RoboDK station: Machine-Tending-Machining-and-Material-Handling-with-Omron-TM12X.rdk

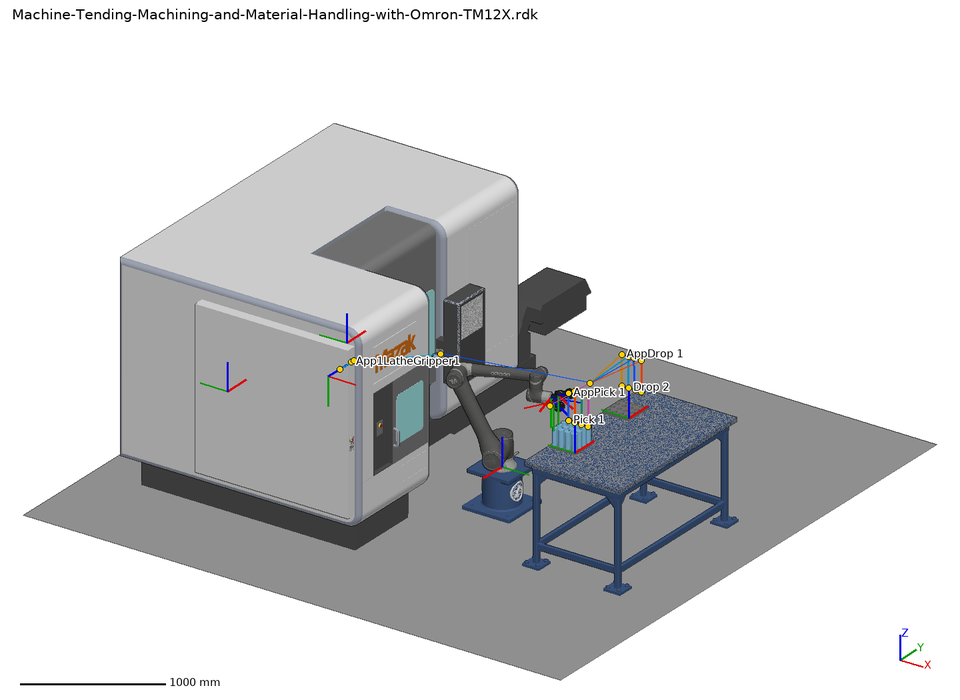
[picture v0: the station drawn from its stored meshes, robots at their saved joint values, targets as dots, program paths as lines]
Station Machine Tending, Machining and Material Handling with Omron TM12X (saved by RoboDK 5.4.3). Poses are relative to the parent item; angles as X-Y-Z fixed-axis rotations.
Station parameters (name, value as stored): TAGS, ['Machine Tending', 'CNC']
  - frame Omron TM12X Base at (300, 0, 70) mm, rotated rx 0 ry 0 rz -90 deg
    - robot Omron TM12X: 6 axes, payload 12 kg, reach 1300 mm, repeatability 0.1 mm, weight 33.3 kg
        modified DH rows (alpha deg, a mm, theta deg, d mm): 0, 0, 0, 165.2; 90, 0, 90, 0; 0, 636.1, 0, 0; 0, 557.9, -90, 156.3; -90, 0, 0, 106; 90, 0, 180, 113.15
        joint limits [-360, -360, -163, -360, -360, -360] to [360, 360, 163, 360, 360, 360]; home [0, 0, 90, -90, 90, 0]; saved at [109.92, -25.7, 113.76, -268.05, -85.72, 0]
      - frame RobotiQ HandE Dual Gripper at (0, 0, -5) mm
        - frame RobotiQ HandE Gripper Base 1 at (50, 0, 40) mm, rotated rx 0 ry 45 rz 0 deg
          - robot RobotiQ HandE Gripper 1: 1 axes
              joint limits [0] to [50]; home [0]; saved at [50]
        - frame RobotiQ HandE Gripper Base 2 at (-50, 0, 40) mm, rotated rx 0 ry -45 rz 0 deg
          - robot RobotiQ HandE Gripper 2: 1 axes
              joint limits [0] to [50]; home [0]; saved at [50]
        - object Hand-E RobotiQ Dual Mounting at (0, 0, 0) mm, size 158.7 x 86.1 x 105 mm, geometry from Hand-E RobotiQ Dual Mounting.step
      - tool Gripper1, TCP at (145, 0, 130) mm, rotated rx 45 ry 0 rz 90 deg
      - tool Gripper2, TCP at (-145, 0, 130) mm, rotated rx -45 ry 0 rz 90 deg
    - object Pedestal H12in (Type 1) at (0, 0, -300) mm, size 400 x 400 x 304.8 mm, geometry from Pedestal-H12in-Type-1.sld
  - frame Mazak Lathe Base at (-1000, 0, 650) mm, rotated rx 0 ry 0 rz 90 deg
    - robot Mazak Lathe: 1 axes
        modified DH rows (alpha deg, a mm, theta deg, d mm): 0, 0, 0, 0 linear
        base shift (0, 0, 0) mm, rotated rx 0 ry 90 rz 0 deg
        joint limits [0] to [700]; home [0]; saved at [0]
    - frame Lathe at (-368.68, -104.77, -79.13) mm, rotated rx -90 ry 0 rz -90 deg
      - target App1LatheGripper1 (Cartesian target) at (-0.18, 0.1, 274.88) mm, rotated rx 0 ry 90 rz 165 deg; joints [287.606, 19.83, 87.712, -318.746, -74.815, 80.984] of Omron TM12X
      - target LatheGripper1 (Cartesian target) at (-0.18, 0.1, 134.88) mm, rotated rx 0 ry 90 rz 165 deg; joints [296.712, 22.07, 84.693, -319.639, -67.09, 75.877] of Omron TM12X
      - target App1LatheGripper2 (Cartesian target) at (-0.18, 0.1, 301.9) mm, rotated rx 0 ry 90 rz 165 deg; joints [285.755, 19.624, 87.976, -318.559, -76.4, 81.971] of Omron TM12X
      - target LatheGripper2 (Cartesian target) at (-0.18, 0.1, 134.88) mm, rotated rx 0 ry 90 rz 165 deg; joints [296.712, 22.07, 84.693, -319.639, -67.09, 75.877] of Omron TM12X
  - frame Input at (1200, -410, 590) mm, rotated rx 0 ry 0 rz 90 deg
    - object Part Matrix at (0, 0, 0) mm, size 220 x 220 x 25 mm, geometry from Part Matrix.step
    - object Part 16 at (27.5, 27.5, -20) mm, size 40 x 40 x 150 mm, geometry from Part.step
    - object Part 15 at (27.5, 82.5, -20) mm, size 40 x 40 x 150 mm, geometry from Part.step
    - object Part 14 at (27.5, 137.5, -20) mm, size 40 x 40 x 150 mm, geometry from Part.step
    - object Part 13 at (27.5, 192.5, -20) mm, size 40 x 40 x 150 mm, geometry from Part.step
    - object Part 12 at (82.5, 27.5, -20) mm, size 40 x 40 x 150 mm, geometry from Part.step
    - object Part 11 at (82.5, 82.5, -20) mm, size 40 x 40 x 150 mm, geometry from Part.step
    - object Part 10 at (82.5, 137.5, -20) mm, size 40 x 40 x 150 mm, geometry from Part.step
    - object Part 9 at (82.5, 192.5, -20) mm, size 40 x 40 x 150 mm, geometry from Part.step
    - object Part 8 at (137.5, 27.5, -20) mm, size 40 x 40 x 150 mm, geometry from Part.step
    - object Part 6 at (137.5, 137.5, -20) mm, size 40 x 40 x 150 mm, geometry from Part.step
    - object Part Done 16 at (27.5, 27.5, -20) mm, size 40.5 x 40.5 x 150 mm, geometry from Part Done.step
    - object Part Done 15 at (27.5, 82.5, -20) mm, size 40.5 x 40.5 x 150 mm, geometry from Part Done.step
    - object Part Done 14 at (27.5, 137.5, -20) mm, size 40.5 x 40.5 x 150 mm, geometry from Part Done.step
    - object Part Done 13 at (27.5, 192.5, -20) mm, size 40.5 x 40.5 x 150 mm, geometry from Part Done.step
    - object Part Done 12 at (82.5, 27.5, -20) mm, size 40.5 x 40.5 x 150 mm, geometry from Part Done.step
    - object Part Done 11 at (82.5, 82.5, -20) mm, size 40.5 x 40.5 x 150 mm, geometry from Part Done.step
    - object Part Done 10 at (82.5, 137.5, -20) mm, size 40.5 x 40.5 x 150 mm, geometry from Part Done.step
    - object Part Done 9 at (82.5, 192.5, -20) mm, size 40.5 x 40.5 x 150 mm, geometry from Part Done.step
    - object Part Done 8 at (137.5, 27.5, -20) mm, size 40.5 x 40.5 x 150 mm, geometry from Part Done.step
    - object Part Done 7 at (137.5, 82.5, -20) mm, size 40.5 x 40.5 x 150 mm, geometry from Part Done.step
    - object Part Done 6 at (137.5, 137.5, -20) mm, size 40.5 x 40.5 x 150 mm, geometry from Part Done.step
    - target Pick 1 (Cartesian target) at (192.5, 192.5, 115) mm, rotated rx 0 ry 90 rz 180 deg; joints [82.224, -15.221, -78.684, -86.096, 127.224, 0] of Omron TM12X
    - target Pick 2 (Cartesian target) at (192.5, 137.5, 115) mm, rotated rx 0 ry 90 rz 180 deg; joints [-125.489, -16.998, -133.125, 63.873, 99.511, 90] of Omron TM12X
    - target Pick 3 (Cartesian target) at (192.5, 82.5, 115) mm, rotated rx 0 ry 90 rz 180 deg; joints [-120.952, -10.605, -128.576, 62.029, 104.048, 90] of Omron TM12X
    - target Pick 4 (Cartesian target) at (192.5, 27.5, 115) mm, rotated rx 0 ry 90 rz 180 deg; joints [-117.466, -4.841, -123.761, 61.08, 107.534, 90] of Omron TM12X
    - target AppPick 1 (Cartesian target) at (192.5, 192.5, 325) mm, rotated rx 0 ry 90 rz 180 deg; joints [82.224, -17.921, -53.195, -108.884, 127.224, 0] of Omron TM12X
    - target AppPick 2 (Cartesian target) at (192.5, 137.5, 355) mm, rotated rx 0 ry 90 rz -180 deg; joints [105.445, 25.882, 38.239, -244.121, -29.555, 0] of Omron TM12X
    - target AppPick 3 (Cartesian target) at (192.5, 82.5, 355) mm, rotated rx 0 ry 90 rz -180 deg; joints [104.438, 34.421, 24.131, -238.551, -30.562, 0] of Omron TM12X
    - target AppPick 4 (Cartesian target) at (192.5, 27.5, 355) mm, rotated rx 0 ry 90 rz -180 deg; joints [105.251, 27.242, 36.106, -243.348, -29.749, 0] of Omron TM12X
    - object Part 5 at (137.5, 192.5, -20) mm, size 40 x 40 x 150 mm, geometry from Part.step
    - object Part Done 5 at (137.5, 192.5, -20) mm, size 40.5 x 40.5 x 150 mm, geometry from Part Done.step
    - object Part 7 at (137.5, 82.5, -20) mm, size 40 x 40 x 150 mm, geometry from Part.step
    - object Part 4 at (192.5, 27.5, -20) mm, rotated rx 0 ry 0 rz -180 deg, size 40 x 40 x 150 mm, geometry from Part.step
    - object Part Done 4 at (192.5, 27.5, -20) mm, rotated rx 0 ry 0 rz 180 deg, size 40.5 x 40.5 x 150 mm, geometry from Part Done.step
    - object Part Done 3 at (192.5, 82.5, -20) mm, rotated rx 0 ry 0 rz -180 deg, size 40.5 x 40.5 x 150 mm, geometry from Part Done.step
    - object Part 3 at (192.5, 82.5, -20) mm, rotated rx 0 ry 0 rz -180 deg, size 40 x 40 x 150 mm, geometry from Part.step
    - object Part 2 at (192.5, 137.5, -20) mm, rotated rx 0 ry 0 rz -180 deg, size 40 x 40 x 150 mm, geometry from Part.step
    - object Part Done 2 at (192.5, 137.5, -20) mm, rotated rx 0 ry 0 rz -180 deg, size 40.5 x 40.5 x 150 mm, geometry from Part Done.step
    - object Part 1 at (192.5, 192.5, -20) mm, rotated rx 0 ry 0 rz -180 deg, size 40 x 40 x 150 mm, geometry from Part.step
    - object Part Done 1 at (192.5, 192.5, -20) mm, rotated rx 0 ry 0 rz -180 deg, size 40.5 x 40.5 x 150 mm, geometry from Part Done.step
  - frame Output at (1200, 230, 600) mm, rotated rx 0 ry 0 rz 90 deg
    - object Part Matrix at (0, 0, 0) mm, size 220 x 220 x 25 mm, geometry from Part Matrix.step
    - target Drop 1 (Cartesian target) at (192.5, 192.5, 115) mm, rotated rx 0 ry 90 rz 0 deg; joints [116.866, 7.231, 87.421, -274.651, -108.134, 0] of Omron TM12X
    - target Drop 2 (Cartesian target) at (192.5, 137.5, 115) mm, rotated rx 0 ry 90 rz 0 deg; joints [114.797, 12.211, 81.48, -273.69, -110.203, 0] of Omron TM12X
    - target Drop 3 (Cartesian target) at (192.5, 82.5, 115) mm, rotated rx 0 ry 90 rz 0 deg; joints [113.02, 17.279, 74.94, -272.218, -111.98, 0] of Omron TM12X
    - target Drop 4 (Cartesian target) at (192.5, 27.5, 115) mm, rotated rx 0 ry 90 rz 0 deg; joints [111.479, 22.52, 67.664, -270.184, -113.521, 0] of Omron TM12X
    - target AppDrop 1 (Cartesian target) at (192.5, 192.5, 355) mm, rotated rx 0 ry 90 rz 0 deg; joints [116.866, 10.453, 58.512, -248.965, -108.134, 0] of Omron TM12X
    - target AppDrop 2 (Cartesian target) at (192.5, 137.5, 355) mm, rotated rx 0 ry 90 rz 0 deg; joints [114.797, 16.092, 51.283, -247.375, -110.203, 0] of Omron TM12X
    - target AppDrop 3 (Cartesian target) at (192.5, 92.5, 355) mm, rotated rx 0 ry 90 rz 0 deg; joints [113.324, 21.121, 44.257, -245.378, -111.676, 0] of Omron TM12X
    - target AppDrop 4 (Cartesian target) at (192.5, 27.5, 355) mm, rotated rx 0 ry 90 rz 0 deg; joints [111.479, 29.696, 30.978, -240.675, -113.521, 0] of Omron TM12X
  - frame World at (-2000, 0, 0) mm, rotated rx 0 ry 0 rz 90 deg
    - target Transition 1 (joint target) at (320.62, -2812.4, 721.26) mm, rotated rx 0 ry 90 rz -75.38 deg; joints [153.89, -25.7, 113.76, -268.06, -85.73, 0] of Omron TM12X
    - target Transition 2 (joint target) at (110.77, -1705.81, 721.22) mm, rotated rx -130.72 ry 89.99 rz -68.7 deg; joints [291.3, -25.7, 113.76, -268.05, -85.72, 0] of Omron TM12X
    - target Gripper1 Open (Cartesian target) at (-535.44, -2699.33, 504.11) mm, rotated rx -90 ry 0 rz 90 deg; joints [50, 0, 0, 0, 0, 0] of RobotiQ HandE Gripper 1
    - target Gripper1 Close (Cartesian target) at (-535.44, -2699.33, 504.11) mm, rotated rx -90 ry 0 rz 90 deg; joints [40, 0, 0, 0, 0, 0] of RobotiQ HandE Gripper 1
    - target Gripper2 Open (Cartesian target) at (-314.73, -2920.04, 504.11) mm, rotated rx -90 ry 0 rz 180 deg; joints [50, 0, 0, 0, 0, 0] of RobotiQ HandE Gripper 2
    - target Gripper2 Close (Cartesian target) at (-314.73, -2920.04, 504.11) mm, rotated rx -90 ry 0 rz 180 deg; joints [40, 0, 0, 0, 0, 0] of RobotiQ HandE Gripper 2
    - target Door1 Open (Cartesian target) at (700, -1000, 650) mm; joints [700, 0, 0, 0, 0, 0] of Mazak Lathe
    - target Door1 Close (Cartesian target) at (0, -1000, 650) mm; joints [0, 0, 0, 0, 0, 0] of Mazak Lathe
    - target Home (joint target) at (-125.05, -2791.35, 721.22) mm, rotated rx -130.72 ry 89.99 rz 109.92 deg; joints [109.92, -25.7, 113.76, -268.05, -85.72, 0] of Omron TM12X
    - object Floor at (250, -1940, -230) mm, size 4500 x 4500 x 0 mm, geometry from Floor (2).sld
    - object Table 1400x800x800mm at (-340, -3360, 570) mm, size 1420 x 820 x 800 mm, geometry from Table-1400x800x800mm.sld
  - folder Mechanism Programs
    - program OpenGripper1 (1 instructions, listed below)
    - program CloseGripper1 (1 instructions, listed below)
    - program OpenGripper2 (1 instructions, listed below)
    - program CloseGripper2 (1 instructions, listed below)
    - program OpenDoor1 (1 instructions, listed below)
    - program CloseDoor1 (1 instructions, listed below)
  - folder PickInput Programs
    - program Pick 1 (6 instructions, listed below)
    - program Pick 2 (6 instructions, listed below)
    - program Pick 3 (6 instructions, listed below)
    - program Pick 4 (6 instructions, listed below)
  - folder DropOutput Programs
    - program Drop 1 (9 instructions, listed below)
    - program Drop 2 (9 instructions, listed below)
    - program Drop 3 (9 instructions, listed below)
    - program Drop 4 (9 instructions, listed below)
  - folder Other Programs
    - program GoHome (3 instructions, listed below)
    - program ReplaceObjects (1 instructions, listed below)
    - program Init (6 instructions, listed below)
    - program PickLatheTransition (4 instructions, listed below)
    - program LathePickTransition (4 instructions, listed below)
  - folder Lath Programs
    - folder Work Programs
      - program Work 1 (3 instructions, listed below)
      - program Work 2 (3 instructions, listed below)
      - program Work 3 (3 instructions, listed below)
      - program Work 4 (3 instructions, listed below)
    - program PickLathe (9 instructions, listed below)
    - program DropLathe (12 instructions, listed below)
  - folder Gripper Programs
    - program Gripper1PickInput (3 instructions, listed below)
    - program Gripper2DropOutput (3 instructions, listed below)
  - program MainProgram (41 instructions, listed below)
  - program Reset (2 instructions, listed below)
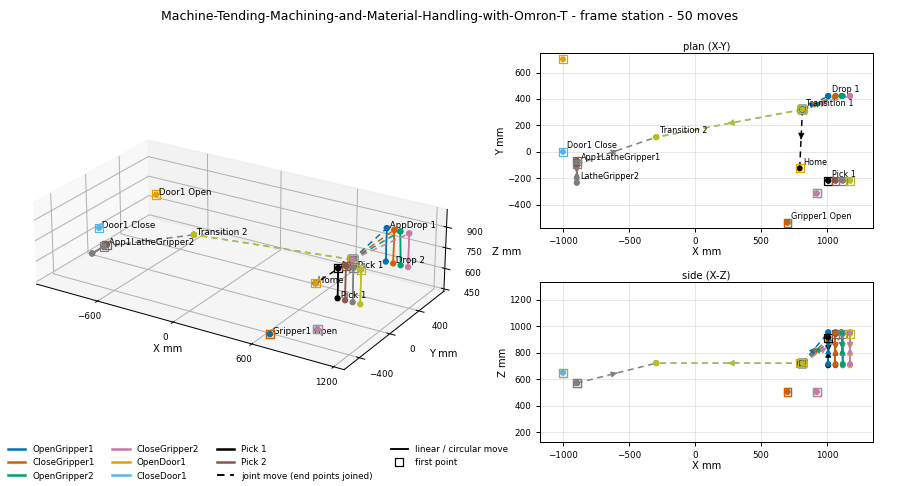
[picture p0: tool path of Machine-Tending-Machining-and-Material-Handling-with-Omron-TM12X.rdk in frame station, 50 of 50 moves have a stored position in this frame; points joined in program order, loops and branches not executed]

--- program OpenGripper1 (robot RobotiQ HandE Gripper 1) ---
  MoveJ (Gripper1 Open)

--- program CloseGripper1 (robot RobotiQ HandE Gripper 1) ---
  MoveJ (Gripper1 Close)

--- program OpenGripper2 (robot RobotiQ HandE Gripper 2) ---
  MoveJ (Gripper2 Open)

--- program CloseGripper2 (robot RobotiQ HandE Gripper 2) ---
  MoveJ (Gripper2 Close)

--- program OpenDoor1 (robot Mazak Lathe) ---
  MoveJ (Door1 Open)

--- program CloseDoor1 (robot Mazak Lathe) ---
  MoveJ (Door1 Close)

--- program Pick 1 (robot Omron TM12X) ---
  Set Ref.: Input
  Set Tool: Gripper1
  MoveJ (AppPick 1)
  MoveL (Pick 1)
  Call Gripper1PickInput
  MoveL (AppPick 1)

--- program Pick 2 (robot Omron TM12X) ---
  Set Ref.: Input
  Set Tool: Gripper1
  MoveJ (AppPick 2)
  MoveL (Pick 2)
  Call Gripper1PickInput
  MoveL (AppPick 2)

--- program Pick 3 (robot Omron TM12X) ---
  Set Ref.: Input
  Set Tool: Gripper1
  MoveJ (AppPick 3)
  MoveL (Pick 3)
  Call Gripper1PickInput
  MoveL (AppPick 3)

--- program Pick 4 (robot Omron TM12X) ---
  Set Ref.: Input
  Set Tool: Gripper1
  MoveJ (AppPick 4)
  MoveL (Pick 4)
  Call Gripper1PickInput
  MoveL (AppPick 4)

--- program Drop 1 (robot Omron TM12X) ---
  Set Ref.: World
  Set Tool: Gripper1
  MoveJ (Transition 1)
  Set Ref.: Output
  Set Tool: Gripper2
  MoveJ (AppDrop 1)
  MoveL (Drop 1)
  Call Gripper2DropOutput
  MoveL (AppDrop 1)

--- program Drop 2 (robot Omron TM12X) ---
  Set Ref.: World
  Set Tool: Gripper1
  MoveJ (Transition 1)
  Set Ref.: Output
  Set Tool: Gripper2
  MoveJ (AppDrop 2)
  MoveL (Drop 2)
  Call Gripper2DropOutput
  MoveL (AppDrop 2)

--- program Drop 3 (robot Omron TM12X) ---
  Set Ref.: World
  Set Tool: Gripper1
  MoveJ (Transition 1)
  Set Ref.: Output
  Set Tool: Gripper2
  MoveJ (AppDrop 3)
  MoveL (Drop 3)
  Call Gripper2DropOutput
  MoveL (AppDrop 3)

--- program Drop 4 (robot Omron TM12X) ---
  Set Ref.: World
  Set Tool: Gripper1
  MoveJ (Transition 1)
  Set Ref.: Output
  Set Tool: Gripper2
  MoveJ (AppDrop 4)
  MoveL (Drop 4)
  Call Gripper2DropOutput
  MoveL (AppDrop 4)

--- program GoHome (robot Omron TM12X) ---
  Set Ref.: World
  Set Tool: Gripper1
  MoveJ (Home)

--- program ReplaceObjects (robot Omron TM12X) ---
  Replace objects

--- program Init (robot Omron TM12X) ---
  Run OpenGripper1
  Run OpenGripper2
  Run CloseDoor1
  Run ReplaceObjects
  Show objects
  Hide objects

--- program PickLatheTransition (robot Omron TM12X) ---
  Set Ref.: World
  Set Tool: Gripper1
  MoveJ (Transition 1)
  MoveJ (Transition 2)

--- program LathePickTransition (robot Omron TM12X) ---
  Set Ref.: World
  Set Tool: Gripper1
  MoveJ (Transition 1)
  MoveJ (Home)

--- program Work 1 (robot Omron TM12X) ---
  Pause 10.0 s
  Show Part Done 1
  Hide Part 1

--- program Work 2 (robot Omron TM12X) ---
  Pause 10.0 s
  Show Part Done 2
  Hide Part 2

--- program Work 3 (robot Omron TM12X) ---
  Pause 10.0 s
  Show Part Done 3
  Hide Part 3

--- program Work 4 (robot Omron TM12X) ---
  Pause 10.0 s
  Show Part Done 4
  Hide Part 4

--- program PickLathe (robot Omron TM12X) ---
  Call OpenDoor1
  Set Ref.: Lathe
  Set Tool: Gripper2
  MoveJ (App1LatheGripper2)
  MoveL (LatheGripper2)
  Call CloseGripper2
  Attach to Gripper2
  Attach to Gripper2
  MoveL (App1LatheGripper2)

--- program DropLathe (robot Omron TM12X) ---
  Call OpenDoor1
  Set Ref.: Lathe
  Set Tool: Gripper1
  MoveJ (App1LatheGripper1)
  MoveL (LatheGripper1)
  Call OpenGripper1
  Detach from Gripper1
  Detach from Gripper1
  MoveJ (App1LatheGripper1)
  Set Ref.: World
  MoveJ (Transition 2)
  Call CloseDoor1

--- program Gripper1PickInput (robot Omron TM12X) ---
  Call CloseGripper1
  Attach to Gripper1
  Attach to Gripper1

--- program Gripper2DropOutput (robot Omron TM12X) ---
  Call OpenGripper2
  Detach from Gripper2
  Detach from Gripper2

--- program MainProgram (robot Omron TM12X) ---
  Call Init
  Call GoHome
  Call Pick 1
  Call PickLatheTransition
  Call DropLathe
  Call LathePickTransition
  Call Pick 2
  Call PickLatheTransition
  Call Work 1
  Call PickLathe
  Call DropLathe
  Call Drop 1
  Call LathePickTransition
  Call Pick 3
  Call PickLatheTransition
  Call Work 2
  Call PickLathe
  Call DropLathe
  Call Drop 2
  Call LathePickTransition
  Call Pick 4
  Call PickLatheTransition
  Call Work 3
  Call PickLathe
  Call DropLathe
  Call Drop 3
  Set Ref.: World
  Set Tool: Gripper1
  MoveJ (Transition 1)
  MoveJ (Transition 2)
  Call Work 4
  Set Ref.: World
  Set Tool: Gripper1
  MoveJ (Transition 2)
  Call PickLathe
  Set Ref.: World
  Set Tool: Gripper1
  MoveJ (Transition 2)
  Call CloseDoor1
  Call Drop 4
  Call GoHome

--- program Reset (robot Omron TM12X) ---
  Call Init
  Call GoHome
